KUKA KRL program: chk_w9_grp5_vac_on.src

&ACCESS RV4
&COMMENT Axor Traseiro Vaccum on
DEF chk_w9_grp5_vac_on( )

; Check Vacuum on gripper AXOR/ATEGO TRASEIRO
;//---- Start User-------

$TIMER[10] = 0
$TIMER_STOP[10] = FALSE

;FOLD WAIT FOR ( IN 504 'Z6.1 - Vacuo Ligado - AXOR ATEGO 903' );%{PE}%R 8.2.20,%MKUKATPBASIS,%CEXT_WAIT_FOR,%VEXT_WAIT_FOR,%P 2:, 4:, 5:$IN, 6:504, 7:Z6.1 - Vacuo Ligado - AXOR ATEGO 903, 9:
WAIT FOR  ( $IN[504] )
;ENDFOLD

$TIMER_STOP[10] = TRUE
$TIMER[10] = 0

;//---- End User---------

END
